SYSTEM System (* System Configuration *)
  (* Standard: 61499-1 *)
  (* Version 0.3, 2003-12-05, JHC, Rockwell Automation, Renamed from NEWSYSTEM. *)
  (* Version 0.2, 2002-11-05, JHC, Rockwell Automation, Fixed missing (empty) FBD in Application. *)
  (* Version 0.1, 2002-01-17, JHC, Rockwell Automation, Minor cleanup *)
  (* Version 0.0, 2000-05-27, JHC, Rockwell Automation *)
  APPLICATION APP1
  END_APPLICATION
  DEVICE STATION_2 : ImageDev(Length := 750, Height := 750)
    RESOURCE image : ImageResource
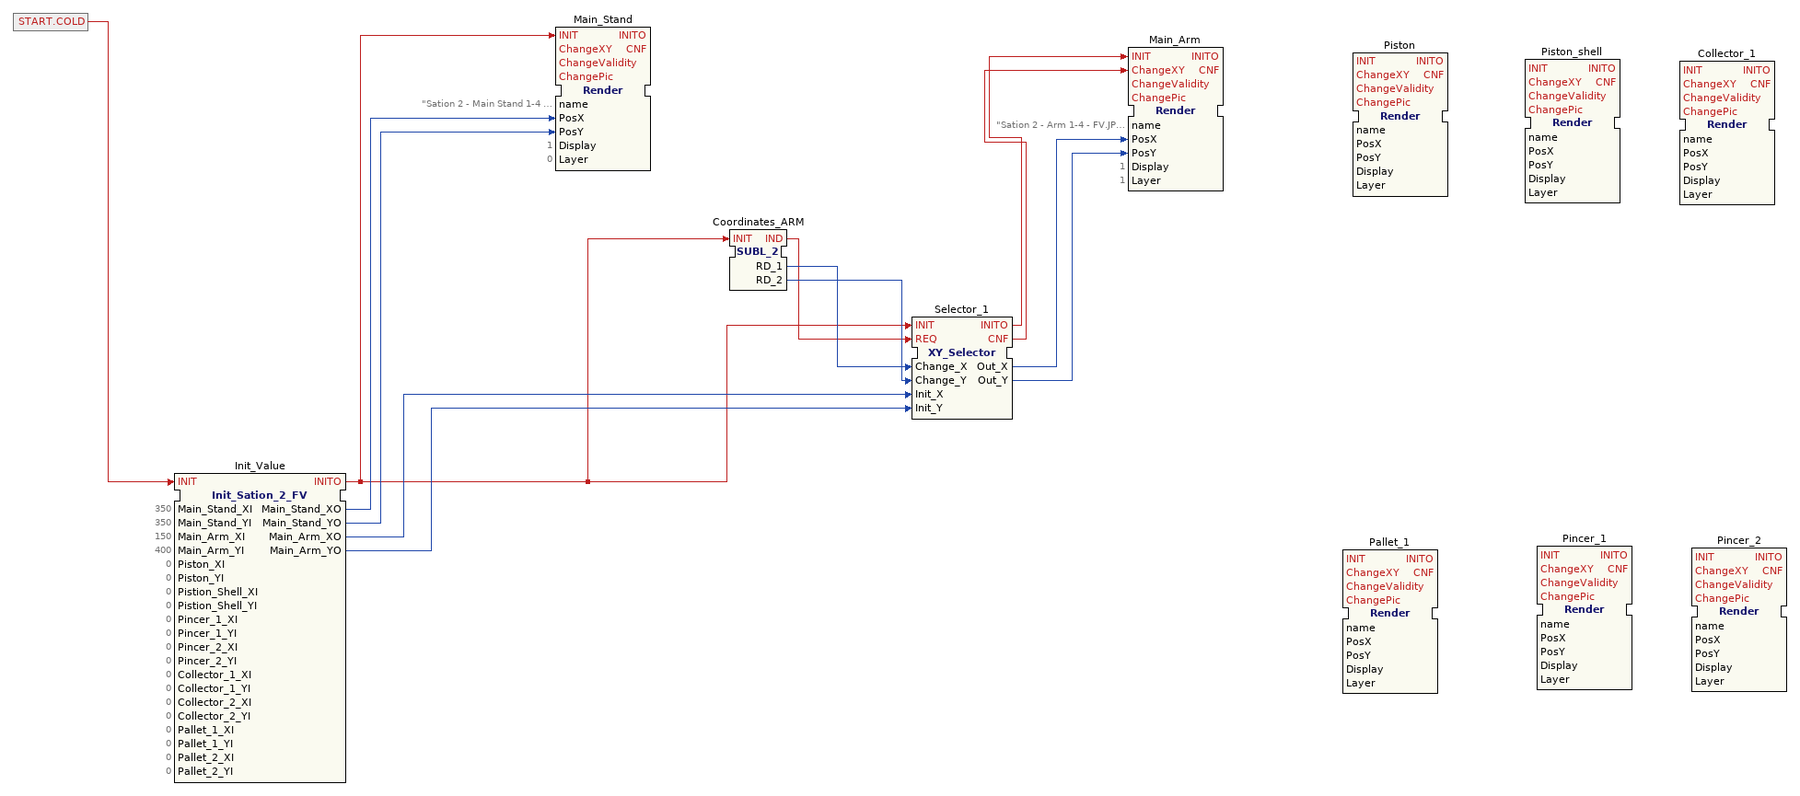
      FBS
        Coordinates_ARM : SUBL_2;
        Main_Stand : Render(Display := 1, Layer := 0, name := "Sation 2 - Main Stand 1-4 - FV.JPG");
        Piston : Render;
        Piston_shell : Render;
        Pincer_1 : Render;
        Pincer_2 : Render;
        Collector_1 : Render;
        Pallet_1 : Render;
        Main_Arm : Render(name := "Sation 2 - Arm 1-4 - FV.JPG", Display := 1, Layer := 1);
        Init_Value : Init_Sation_2_FV(Main_Stand_XI := 350, Main_Stand_YI := 350, Main_Arm_XI := 150, Main_Arm_YI := 400, Piston_XI := 0, Piston_YI := 0, Pistion_Shell_XI := 0, Pistion_Shell_YI := 0, Pincer_1_XI := 0, Pincer_1_YI := 0, Pincer_2_XI := 0, Pincer_2_YI := 0, Collector_1_XI := 0, Collector_1_YI := 0, Collector_2_XI := 0, Collector_2_YI := 0, Pallet_1_XI := 0, Pallet_1_YI := 0, Pallet_2_XI := 0, Pallet_2_YI := 0);
        Selector_1 : XY_Selector;
      END_FBS
      EVENT_CONNECTIONS
        Init_Value.INITO TO Main_Stand.INIT;
        START.COLD TO Init_Value.INIT;
        Init_Value.INITO TO Coordinates_ARM.INIT;
        Selector_1.INITO TO Main_Arm.INIT;
        Init_Value.INITO TO Selector_1.INIT;
        Coordinates_ARM.IND TO Selector_1.REQ;
        Selector_1.CNF TO Main_Arm.ChangeXY;
      END_CONNECTIONS
      DATA_CONNECTIONS
        Selector_1.Out_X TO Main_Arm.PosX;
        Selector_1.Out_Y TO Main_Arm.PosY;
        Coordinates_ARM.RD_1 TO Selector_1.Change_X;
        Coordinates_ARM.RD_2 TO Selector_1.Change_Y;
        Init_Value.Main_Stand_XO TO Main_Stand.PosX;
        Init_Value.Main_Stand_YO TO Main_Stand.PosY;
        Init_Value.Main_Arm_XO TO Selector_1.Init_X;
        Init_Value.Main_Arm_YO TO Selector_1.Init_Y;
      END_CONNECTIONS
    END_RESOURCE
  END_DEVICE
  DEVICE Frame : FRAME_DEVICE(BOUNDS := [0,301,300,100], GRID := [1,1])
    RESOURCE panel : PANEL_RESOURCE
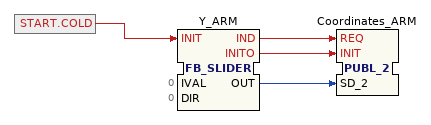
      FBS
        Y_ARM : FB_SLIDER(IVAL := 0, DIR := 0);
        Coordinates_ARM : PUBL_2;
      END_FBS
      EVENT_CONNECTIONS
        Y_ARM.IND TO Coordinates_ARM.REQ;
        Y_ARM.INITO TO Coordinates_ARM.INIT;
        START.COLD TO Y_ARM.INIT;
      END_CONNECTIONS
      DATA_CONNECTIONS
        Y_ARM.OUT TO Coordinates_ARM.SD_2;
      END_CONNECTIONS
    END_RESOURCE
  END_DEVICE
END_SYSTEM
